// Alias for the error object.
TYPE T_Error : FB_Error; END_TYPE

(* stored: Version 1.1.0.1
   DUT T_Error: Id {c1df8a4e-e064-0857-16ff-9a0f6aacee61} *)
